Fanuc TP program (LS listing): DISTI_CADC_V7.LS

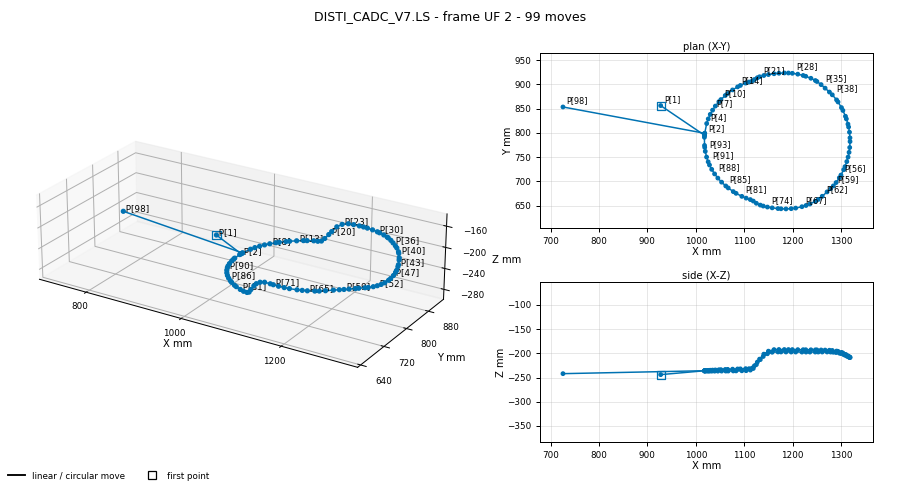
[picture p0: tool path of DISTI_CADC_V7.LS in frame UF 2, 99 of 99 moves have a stored position in this frame; points joined in program order, loops and branches not executed]
/PROG  DISTI_CADC_V7
/ATTR
OWNER		= MNEDITOR;
COMMENT		= "WeldPRO Auto-Gen";
PROG_SIZE	= 7109;
CREATE		= DATE 26-07-21  TIME 18:28:40;
MODIFIED	= DATE 26-07-21  TIME 18:47:32;
FILE_NAME	= DISTI_CA;
VERSION		= 0;
LINE_COUNT	= 113;
MEMORY_SIZE	= 7429;
PROTECT		= READ_WRITE;
TCD:  STACK_SIZE	= 0,
      TASK_PRIORITY	= 50,
      TIME_SLICE	= 0,
      BUSY_LAMP_OFF	= 0,
      ABORT_REQUEST	= 0,
      PAUSE_REQUEST	= 0;
DEFAULT_GROUP	= 1,*,*,*,*;
CONTROL_CODE	= 00000000 00000000;
/APPL
/MN
   1:  !WeldPRO Auto-Generated TPP ;
   2:  !Tor XL_176 _2, Feature1 ;
   3:   ;
   4:  UFRAME_NUM=2 ;
   5:  UTOOL_NUM=2 ;
   6:L P[1] 100mm/sec FINE    ;
   7:   ;
   8:  !Segment1 ;
   9:L P[2] 100mm/sec FINE    ;
  10:  CALL LASER_OFF    ;
  11:   ;
  12:L P[99] R[23:moving]mm/sec CNT100    ;
  13:   ;
  14:L P[3] R[23:moving]mm/sec CNT100    ;
  15:L P[4] R[23:moving]mm/sec CNT100    ;
  16:L P[5] R[23:moving]mm/sec CNT100    ;
  17:L P[6] R[23:moving]mm/sec CNT100    ;
  18:L P[7] R[23:moving]mm/sec CNT100    ;
  19:L P[8] R[23:moving]mm/sec CNT100    ;
  20:L P[9] R[23:moving]mm/sec CNT100    ;
  21:L P[10] R[23:moving]mm/sec CNT100    ;
  22:L P[11] R[23:moving]mm/sec CNT100    ;
  23:L P[12] R[23:moving]mm/sec CNT100    ;
  24:L P[13] R[23:moving]mm/sec CNT100    ;
  25:L P[14] R[23:moving]mm/sec CNT100    ;
  26:L P[15] R[23:moving]mm/sec CNT100    ;
  27:L P[16] R[23:moving]mm/sec CNT100    ;
  28:L P[17] R[23:moving]mm/sec CNT100    ;
  29:L P[18] R[23:moving]mm/sec CNT100    ;
  30:L P[19] R[23:moving]mm/sec CNT100    ;
  31:L P[20] R[23:moving]mm/sec CNT100    ;
  32:L P[21] R[23:moving]mm/sec CNT100    ;
  33:L P[22] R[23:moving]mm/sec CNT100    ;
  34:L P[23] R[23:moving]mm/sec CNT100    ;
  35:L P[24] R[23:moving]mm/sec CNT100    ;
  36:L P[25] R[23:moving]mm/sec CNT100    ;
  37:L P[26] R[23:moving]mm/sec CNT100    ;
  38:L P[27] R[23:moving]mm/sec CNT100    ;
  39:L P[28] R[23:moving]mm/sec CNT100    ;
  40:L P[29] R[23:moving]mm/sec CNT100    ;
  41:L P[30] R[23:moving]mm/sec CNT100    ;
  42:L P[31] R[23:moving]mm/sec CNT100    ;
  43:L P[32] R[23:moving]mm/sec CNT100    ;
  44:L P[33] R[23:moving]mm/sec CNT100    ;
  45:L P[34] R[23:moving]mm/sec CNT100    ;
  46:L P[35] R[23:moving]mm/sec CNT100    ;
  47:L P[36] R[23:moving]mm/sec CNT100    ;
  48:L P[37] R[23:moving]mm/sec CNT100    ;
  49:L P[38] R[23:moving]mm/sec CNT100    ;
  50:L P[39] R[23:moving]mm/sec CNT100    ;
  51:L P[40] R[23:moving]mm/sec CNT100    ;
  52:L P[41] R[23:moving]mm/sec CNT100    ;
  53:L P[42] R[23:moving]mm/sec CNT100    ;
  54:L P[43] R[23:moving]mm/sec CNT100    ;
  55:L P[44] R[23:moving]mm/sec CNT100    ;
  56:L P[45] R[23:moving]mm/sec CNT100    ;
  57:L P[46] R[23:moving]mm/sec CNT100    ;
  58:L P[47] R[23:moving]mm/sec CNT100    ;
  59:L P[48] R[23:moving]mm/sec CNT100    ;
  60:L P[49] R[23:moving]mm/sec CNT100    ;
  61:L P[50] R[23:moving]mm/sec CNT100    ;
  62:L P[51] R[23:moving]mm/sec CNT100    ;
  63:L P[52] R[23:moving]mm/sec CNT100    ;
  64:L P[53] R[23:moving]mm/sec CNT100    ;
  65:L P[54] R[23:moving]mm/sec CNT100    ;
  66:L P[55] R[23:moving]mm/sec CNT100    ;
  67:L P[56] R[23:moving]mm/sec CNT100    ;
  68:L P[57] R[23:moving]mm/sec CNT100    ;
  69:L P[58] R[23:moving]mm/sec CNT100    ;
  70:L P[59] R[23:moving]mm/sec CNT100    ;
  71:L P[60] R[23:moving]mm/sec CNT100    ;
  72:L P[61] R[23:moving]mm/sec CNT100    ;
  73:L P[62] R[23:moving]mm/sec CNT100    ;
  74:L P[63] R[23:moving]mm/sec CNT100    ;
  75:L P[64] R[23:moving]mm/sec CNT100    ;
  76:L P[65] R[23:moving]mm/sec CNT100    ;
  77:L P[66] R[23:moving]mm/sec CNT100    ;
  78:L P[67] R[23:moving]mm/sec CNT100    ;
  79:L P[68] R[23:moving]mm/sec CNT100    ;
  80:L P[69] R[23:moving]mm/sec CNT100    ;
  81:L P[70] R[23:moving]mm/sec CNT100    ;
  82:L P[71] R[23:moving]mm/sec CNT100    ;
  83:L P[72] R[23:moving]mm/sec CNT100    ;
  84:L P[73] R[23:moving]mm/sec CNT100    ;
  85:L P[74] R[23:moving]mm/sec CNT100    ;
  86:L P[75] R[23:moving]mm/sec CNT100    ;
  87:L P[76] R[23:moving]mm/sec CNT100    ;
  88:L P[77] R[23:moving]mm/sec CNT100    ;
  89:L P[78] R[23:moving]mm/sec CNT100    ;
  90:L P[79] R[23:moving]mm/sec CNT100    ;
  91:L P[80] R[23:moving]mm/sec CNT100    ;
  92:L P[81] R[23:moving]mm/sec CNT100    ;
  93:L P[82] R[23:moving]mm/sec CNT100    ;
  94:L P[83] R[23:moving]mm/sec CNT100    ;
  95:L P[84] R[23:moving]mm/sec CNT100    ;
  96:L P[85] R[23:moving]mm/sec CNT100    ;
  97:L P[86] R[23:moving]mm/sec CNT100    ;
  98:L P[87] R[23:moving]mm/sec CNT100    ;
  99:L P[88] R[23:moving]mm/sec CNT100    ;
 100:L P[89] R[23:moving]mm/sec CNT100    ;
 101:L P[90] R[23:moving]mm/sec CNT100    ;
 102:L P[91] R[23:moving]mm/sec CNT100    ;
 103:L P[92] R[23:moving]mm/sec CNT100    ;
 104:L P[93] R[23:moving]mm/sec CNT100    ;
 105:L P[94] R[23:moving]mm/sec CNT100    ;
 106:L P[95] R[23:moving]mm/sec CNT100    ;
 107:L P[96] R[23:moving]mm/sec CNT100    ;
 108:L P[97] R[23:moving]mm/sec FINE    ;
 109:  CALL LASER_OFF    ;
 110:   ;
 111:  !Feature Retreat ;
 112:L P[98] 100mm/sec FINE    ;
 113:  CALL ROTATE    ;
/POS
P[1]{
   GP1:
	UF : 2, UT : 2,		CONFIG : 'F D T, 0, 0, 0',
	X =   927.346  mm,	Y =   856.354  mm,	Z =  -244.034  mm,
	W =  -106.482 deg,	P =   -15.198 deg,	R =    86.345 deg
};
P[2]{
   GP1:
	UF : 2, UT : 2,		CONFIG : 'F D T, 0, 0, 0',
	X =  1017.889  mm,	Y =   795.080  mm,	Z =  -236.060  mm,
	W =  -106.491 deg,	P =   -15.193 deg,	R =    86.327 deg
};
P[3]{
   GP1:
	UF : 2, UT : 2,		CONFIG : 'F D T, 0, 0, 0',
	X =  1018.277  mm,	Y =   799.191  mm,	Z =  -235.971  mm,
	W =  -106.495 deg,	P =   -15.194 deg,	R =    86.332 deg
};
P[4]{
   GP1:
	UF : 2, UT : 2,		CONFIG : 'F D T, 0, 0, 0',
	X =  1022.296  mm,	Y =   819.337  mm,	Z =  -235.500  mm,
	W =  -106.425 deg,	P =   -15.445 deg,	R =    76.281 deg
};
P[5]{
   GP1:
	UF : 2, UT : 2,		CONFIG : 'F D T, 0, 0, 0',
	X =  1025.521  mm,	Y =   828.846  mm,	Z =  -235.241  mm,
	W =  -106.381 deg,	P =   -15.559 deg,	R =    71.464 deg
};
P[6]{
   GP1:
	UF : 2, UT : 2,		CONFIG : 'F D T, 0, 0, 0',
	X =  1029.666  mm,	Y =   838.199  mm,	Z =  -234.962  mm,
	W =  -106.310 deg,	P =   -15.698 deg,	R =    65.272 deg
};
P[7]{
   GP1:
	UF : 2, UT : 2,		CONFIG : 'F D T, 0, 0, 0',
	X =  1034.494  mm,	Y =   846.923  mm,	Z =  -234.669  mm,
	W =  -106.251 deg,	P =   -15.795 deg,	R =    60.811 deg
};
P[8]{
   GP1:
	UF : 2, UT : 2,		CONFIG : 'F D T, 0, 0, 0',
	X =  1040.175  mm,	Y =   855.353  mm,	Z =  -234.358  mm,
	W =  -106.174 deg,	P =   -15.897 deg,	R =    55.794 deg
};
P[9]{
   GP1:
	UF : 2, UT : 2,		CONFIG : 'F D T, 0, 0, 0',
	X =  1047.451  mm,	Y =   864.304  mm,	Z =  -233.991  mm,
	W =  -106.090 deg,	P =   -15.988 deg,	R =    50.970 deg
};
P[10]{
   GP1:
	UF : 2, UT : 2,		CONFIG : 'F D T, 0, 0, 0',
	X =  1051.689  mm,	Y =   868.820  mm,	Z =  -233.793  mm,
	W =  -106.027 deg,	P =   -16.056 deg,	R =    47.314 deg
};
P[11]{
   GP1:
	UF : 2, UT : 2,		CONFIG : 'F D T, 0, 0, 0',
	X =  1060.630  mm,	Y =   877.184  mm,	Z =  -233.387  mm,
	W =  -105.939 deg,	P =   -16.126 deg,	R =    42.935 deg
};
P[12]{
   GP1:
	UF : 2, UT : 2,		CONFIG : 'F D T, 0, 0, 0',
	X =  1065.640  mm,	Y =   881.308  mm,	Z =  -233.171  mm,
	W =  -105.872 deg,	P =   -16.175 deg,	R =    39.733 deg
};
P[13]{
   GP1:
	UF : 2, UT : 2,		CONFIG : 'F D T, 0, 0, 0',
	X =  1075.744  mm,	Y =   888.688  mm,	Z =  -232.750  mm,
	W =  -105.783 deg,	P =   -16.243 deg,	R =    35.484 deg
};
P[14]{
   GP1:
	UF : 2, UT : 2,		CONFIG : 'F D T, 0, 0, 0',
	X =  1086.136  mm,	Y =   894.999  mm,	Z =  -232.338  mm,
	W =  -105.683 deg,	P =   -16.290 deg,	R =    31.072 deg
};
P[15]{
   GP1:
	UF : 2, UT : 2,		CONFIG : 'F D T, 0, 0, 0',
	X =  1091.851  mm,	Y =   897.963  mm,	Z =  -232.125  mm,
	W =  -105.584 deg,	P =   -16.329 deg,	R =    26.914 deg
};
P[16]{
   GP1:
	UF : 2, UT : 2,		CONFIG : 'F D T, 0, 0, 0',
	X =  1102.710  mm,	Y =   902.806  mm,	Z =  -231.724  mm,
	W =  -105.545 deg,	P =   -16.341 deg,	R =    25.103 deg
};
P[17]{
   GP1:
	UF : 2, UT : 2,		CONFIG : 'F D T, 0, 0, 0',
	X =  1109.763  mm,	Y =   905.007  mm,	Z =  -231.762  mm,
	W =  -115.468 deg,	P =   -16.090 deg,	R =    30.046 deg
};
P[18]{
   GP1:
	UF : 2, UT : 2,		CONFIG : 'F D T, 0, 0, 0',
	X =  1116.013  mm,	Y =   906.877  mm,	Z =  -230.586  mm,
	W =  -126.721 deg,	P =   -15.366 deg,	R =    26.538 deg
};
P[19]{
   GP1:
	UF : 2, UT : 2,		CONFIG : 'F D T, 0, 0, 0',
	X =  1120.858  mm,	Y =   910.112  mm,	Z =  -225.766  mm,
	W =  -119.393 deg,	P =   -15.981 deg,	R =    16.221 deg
};
P[20]{
   GP1:
	UF : 2, UT : 2,		CONFIG : 'F D T, 0, 0, 0',
	X =  1126.832  mm,	Y =   913.808  mm,	Z =  -218.133  mm,
	W =  -115.329 deg,	P =   -16.208 deg,	R =    11.788 deg
};
P[21]{
   GP1:
	UF : 2, UT : 2,		CONFIG : 'F D T, 0, 0, 0',
	X =  1131.495  mm,	Y =   915.872  mm,	Z =  -212.049  mm,
	W =  -112.690 deg,	P =   -16.313 deg,	R =     9.687 deg
};
P[22]{
   GP1:
	UF : 2, UT : 2,		CONFIG : 'F D T, 0, 0, 0',
	X =  1140.206  mm,	Y =   918.445  mm,	Z =  -201.776  mm,
	W =  -110.089 deg,	P =   -16.384 deg,	R =     9.676 deg
};
P[23]{
   GP1:
	UF : 2, UT : 2,		CONFIG : 'F D T, 0, 0, 0',
	X =  1149.741  mm,	Y =   920.397  mm,	Z =  -195.589  mm,
	W =  -107.448 deg,	P =   -16.428 deg,	R =     8.430 deg
};
P[24]{
   GP1:
	UF : 2, UT : 2,		CONFIG : 'F D T, 0, 0, 0',
	X =  1161.315  mm,	Y =   922.076  mm,	Z =  -192.410  mm,
	W =  -105.451 deg,	P =   -16.442 deg,	R =     6.850 deg
};
P[25]{
   GP1:
	UF : 2, UT : 2,		CONFIG : 'F D T, 0, 0, 0',
	X =  1171.380  mm,	Y =   923.106  mm,	Z =  -192.191  mm,
	W =  -104.865 deg,	P =   -16.444 deg,	R =     5.674 deg
};
P[26]{
   GP1:
	UF : 2, UT : 2,		CONFIG : 'F D T, 0, 0, 0',
	X =  1182.566  mm,	Y =   923.704  mm,	Z =  -192.249  mm,
	W =  -104.885 deg,	P =   -16.444 deg,	R =     3.732 deg
};
P[27]{
   GP1:
	UF : 2, UT : 2,		CONFIG : 'F D T, 0, 0, 0',
	X =  1191.043  mm,	Y =   923.608  mm,	Z =  -192.305  mm,
	W =  -104.928 deg,	P =   -16.440 deg,	R =     -.482 deg
};
P[28]{
   GP1:
	UF : 2, UT : 2,		CONFIG : 'F D T, 0, 0, 0',
	X =  1199.100  mm,	Y =   922.988  mm,	Z =  -192.368  mm,
	W =  -104.977 deg,	P =   -16.425 deg,	R =    -5.295 deg
};
P[29]{
   GP1:
	UF : 2, UT : 2,		CONFIG : 'F D T, 0, 0, 0',
	X =  1210.327  mm,	Y =   921.245  mm,	Z =  -192.471  mm,
	W =  -105.026 deg,	P =   -16.401 deg,	R =   -10.039 deg
};
P[30]{
   GP1:
	UF : 2, UT : 2,		CONFIG : 'F D T, 0, 0, 0',
	X =  1221.437  mm,	Y =   918.518  mm,	Z =  -192.590  mm,
	W =  -105.069 deg,	P =   -16.371 deg,	R =   -14.284 deg
};
P[31]{
   GP1:
	UF : 2, UT : 2,		CONFIG : 'F D T, 0, 0, 0',
	X =  1226.752  mm,	Y =   916.839  mm,	Z =  -192.653  mm,
	W =  -105.112 deg,	P =   -16.334 deg,	R =   -18.515 deg
};
P[32]{
   GP1:
	UF : 2, UT : 2,		CONFIG : 'F D T, 0, 0, 0',
	X =  1237.398  mm,	Y =   912.751  mm,	Z =  -192.794  mm,
	W =  -105.156 deg,	P =   -16.287 deg,	R =   -22.931 deg
};
P[33]{
   GP1:
	UF : 2, UT : 2,		CONFIG : 'F D T, 0, 0, 0',
	X =  1246.694  mm,	Y =   908.067  mm,	Z =  -192.936  mm,
	W =  -105.219 deg,	P =   -16.204 deg,	R =   -29.417 deg
};
P[34]{
   GP1:
	UF : 2, UT : 2,		CONFIG : 'F D T, 0, 0, 0',
	X =  1249.746  mm,	Y =   906.136  mm,	Z =  -192.994  mm,
	W =  -105.326 deg,	P =   -16.106 deg,	R =   -35.234 deg
};
P[35]{
   GP1:
	UF : 2, UT : 2,		CONFIG : 'F D T, 0, 0, 0',
	X =  1258.465  mm,	Y =   899.675  mm,	Z =  -193.157  mm,
	W =  -105.307 deg,	P =   -16.055 deg,	R =   -38.974 deg
};
P[36]{
   GP1:
	UF : 2, UT : 2,		CONFIG : 'F D T, 0, 0, 0',
	X =  1266.694  mm,	Y =   892.374  mm,	Z =  -193.348  mm,
	W =  -105.304 deg,	P =   -16.061 deg,	R =   -38.624 deg
};
P[37]{
   GP1:
	UF : 2, UT : 2,		CONFIG : 'F D T, 0, 0, 0',
	X =  1275.636  mm,	Y =   884.289  mm,	Z =  -193.707  mm,
	W =  -105.460 deg,	P =   -15.949 deg,	R =   -44.737 deg
};
P[38]{
   GP1:
	UF : 2, UT : 2,		CONFIG : 'F D T, 0, 0, 0',
	X =  1281.534  mm,	Y =   878.597  mm,	Z =  -194.154  mm,
	W =  -105.652 deg,	P =   -15.892 deg,	R =   -47.603 deg
};
P[39]{
   GP1:
	UF : 2, UT : 2,		CONFIG : 'F D T, 0, 0, 0',
	X =  1290.405  mm,	Y =   868.154  mm,	Z =  -195.366  mm,
	W =  -106.194 deg,	P =   -15.794 deg,	R =   -52.149 deg
};
P[40]{
   GP1:
	UF : 2, UT : 2,		CONFIG : 'F D T, 0, 0, 0',
	X =  1293.358  mm,	Y =   863.881  mm,	Z =  -196.009  mm,
	W =  -106.906 deg,	P =   -15.690 deg,	R =   -56.548 deg
};
P[41]{
   GP1:
	UF : 2, UT : 2,		CONFIG : 'F D T, 0, 0, 0',
	X =  1300.478  mm,	Y =   852.200  mm,	Z =  -198.134  mm,
	W =  -107.559 deg,	P =   -15.603 deg,	R =   -60.015 deg
};
P[42]{
   GP1:
	UF : 2, UT : 2,		CONFIG : 'F D T, 0, 0, 0',
	X =  1303.428  mm,	Y =   846.403  mm,	Z =  -199.394  mm,
	W =  -108.250 deg,	P =   -15.507 deg,	R =   -63.574 deg
};
P[43]{
   GP1:
	UF : 2, UT : 2,		CONFIG : 'F D T, 0, 0, 0',
	X =  1308.723  mm,	Y =   834.279  mm,	Z =  -202.322  mm,
	W =  -109.123 deg,	P =   -15.380 deg,	R =   -68.091 deg
};
P[44]{
   GP1:
	UF : 2, UT : 2,		CONFIG : 'F D T, 0, 0, 0',
	X =  1310.604  mm,	Y =   828.898  mm,	Z =  -203.468  mm,
	W =  -109.894 deg,	P =   -15.253 deg,	R =   -72.476 deg
};
P[45]{
   GP1:
	UF : 2, UT : 2,		CONFIG : 'F D T, 0, 0, 0',
	X =  1313.867  mm,	Y =   818.113  mm,	Z =  -205.461  mm,
	W =  -110.258 deg,	P =   -15.184 deg,	R =   -74.873 deg
};
P[46]{
   GP1:
	UF : 2, UT : 2,		CONFIG : 'F D T, 0, 0, 0',
	X =  1315.235  mm,	Y =   812.168  mm,	Z =  -206.340  mm,
	W =  -110.625 deg,	P =   -15.098 deg,	R =   -77.924 deg
};
P[47]{
   GP1:
	UF : 2, UT : 2,		CONFIG : 'F D T, 0, 0, 0',
	X =  1317.027  mm,	Y =   801.431  mm,	Z =  -207.574  mm,
	W =  -111.046 deg,	P =   -14.958 deg,	R =   -82.908 deg
};
P[48]{
   GP1:
	UF : 2, UT : 2,		CONFIG : 'F D T, 0, 0, 0',
	X =  1318.033  mm,	Y =   789.801  mm,	Z =  -208.385  mm,
	W =  -111.160 deg,	P =   -14.266 deg,	R =   -88.178 deg
};
P[49]{
   GP1:
	UF : 2, UT : 2,		CONFIG : 'F D T, 0, 0, 0',
	X =  1318.168  mm,	Y =   782.182  mm,	Z =  -208.610  mm,
	W =  -111.104 deg,	P =   -14.627 deg,	R =   -91.603 deg
};
P[50]{
   GP1:
	UF : 2, UT : 2,		CONFIG : 'F D T, 0, 0, 0',
	X =  1317.501  mm,	Y =   769.857  mm,	Z =  -208.488  mm,
	W =  -110.785 deg,	P =   -15.101 deg,	R =   -96.403 deg
};
P[51]{
   GP1:
	UF : 2, UT : 2,		CONFIG : 'F D T, 0, 0, 0',
	X =  1316.168  mm,	Y =   759.918  mm,	Z =  -207.950  mm,
	W =  -110.276 deg,	P =   -14.535 deg,	R =  -100.836 deg
};
P[52]{
   GP1:
	UF : 2, UT : 2,		CONFIG : 'F D T, 0, 0, 0',
	X =  1314.124  mm,	Y =   750.096  mm,	Z =  -207.025  mm,
	W =  -109.635 deg,	P =   -14.447 deg,	R =  -105.265 deg
};
P[53]{
   GP1:
	UF : 2, UT : 2,		CONFIG : 'F D T, 0, 0, 0',
	X =  1311.503  mm,	Y =   740.771  mm,	Z =  -205.798  mm,
	W =  -109.103 deg,	P =   -14.384 deg,	R =  -108.504 deg
};
P[54]{
   GP1:
	UF : 2, UT : 2,		CONFIG : 'F D T, 0, 0, 0',
	X =  1307.757  mm,	Y =   730.358  mm,	Z =  -204.011  mm,
	W =  -108.392 deg,	P =   -14.307 deg,	R =  -112.625 deg
};
P[55]{
   GP1:
	UF : 2, UT : 2,		CONFIG : 'F D T, 0, 0, 0',
	X =  1305.065  mm,	Y =   724.102  mm,	Z =  -202.728  mm,
	W =  -107.773 deg,	P =   -14.241 deg,	R =  -116.139 deg
};
P[56]{
   GP1:
	UF : 2, UT : 2,		CONFIG : 'F D T, 0, 0, 0',
	X =  1299.418  mm,	Y =   712.954  mm,	Z =  -200.557  mm,
	W =  -106.932 deg,	P =   -14.149 deg,	R =  -121.162 deg
};
P[57]{
   GP1:
	UF : 2, UT : 2,		CONFIG : 'F D T, 0, 0, 0',
	X =  1296.056  mm,	Y =   707.282  mm,	Z =  -199.652  mm,
	W =  -106.269 deg,	P =   -14.066 deg,	R =  -125.698 deg
};
P[58]{
   GP1:
	UF : 2, UT : 2,		CONFIG : 'F D T, 0, 0, 0',
	X =  1289.374  mm,	Y =   697.456  mm,	Z =  -198.422  mm,
	W =  -105.781 deg,	P =   -13.988 deg,	R =  -130.143 deg
};
P[59]{
   GP1:
	UF : 2, UT : 2,		CONFIG : 'F D T, 0, 0, 0',
	X =  1283.723  mm,	Y =   690.590  mm,	Z =  -197.821  mm,
	W =  -105.502 deg,	P =   -13.914 deg,	R =  -134.519 deg
};
P[60]{
   GP1:
	UF : 2, UT : 2,		CONFIG : 'F D T, 0, 0, 0',
	X =  1278.164  mm,	Y =   684.885  mm,	Z =  -197.494  mm,
	W =  -105.438 deg,	P =   -13.851 deg,	R =  -138.498 deg
};
P[61]{
   GP1:
	UF : 2, UT : 2,		CONFIG : 'F D T, 0, 0, 0',
	X =  1270.775  mm,	Y =   678.212  mm,	Z =  -197.291  mm,
	W =  -105.428 deg,	P =   -13.829 deg,	R =  -139.977 deg
};
P[62]{
   GP1:
	UF : 2, UT : 2,		CONFIG : 'F D T, 0, 0, 0',
	X =  1260.749  mm,	Y =   669.204  mm,	Z =  -197.348  mm,
	W =  -105.443 deg,	P =   -13.863 deg,	R =  -137.727 deg
};
P[63]{
   GP1:
	UF : 2, UT : 2,		CONFIG : 'F D T, 0, 0, 0',
	X =  1252.575  mm,	Y =   662.699  mm,	Z =  -197.405  mm,
	W =  -105.373 deg,	P =   -13.729 deg,	R =  -147.436 deg
};
P[64]{
   GP1:
	UF : 2, UT : 2,		CONFIG : 'F D T, 0, 0, 0',
	X =  1246.362  mm,	Y =   658.782  mm,	Z =  -197.421  mm,
	W =  -105.298 deg,	P =   -13.637 deg,	R =  -156.529 deg
};
P[65]{
   GP1:
	UF : 2, UT : 2,		CONFIG : 'F D T, 0, 0, 0',
	X =  1235.369  mm,	Y =   653.232  mm,	Z =  -197.454  mm,
	W =  -105.278 deg,	P =   -13.619 deg,	R =  -158.873 deg
};
P[66]{
   GP1:
	UF : 2, UT : 2,		CONFIG : 'F D T, 0, 0, 0',
	X =  1227.306  mm,	Y =   650.188  mm,	Z =  -197.457  mm,
	W =  -105.242 deg,	P =   -13.593 deg,	R =  -162.872 deg
};
P[67]{
   GP1:
	UF : 2, UT : 2,		CONFIG : 'F D T, 0, 0, 0',
	X =  1218.912  mm,	Y =   647.653  mm,	Z =  -197.449  mm,
	W =  -105.204 deg,	P =   -13.573 deg,	R =  -166.917 deg
};
P[68]{
   GP1:
	UF : 2, UT : 2,		CONFIG : 'F D T, 0, 0, 0',
	X =  1205.982  mm,	Y =   644.800  mm,	Z =  -197.421  mm,
	W =  -105.160 deg,	P =   -13.560 deg,	R =  -171.451 deg
};
P[69]{
   GP1:
	UF : 2, UT : 2,		CONFIG : 'F D T, 0, 0, 0',
	X =  1196.678  mm,	Y =   643.604  mm,	Z =  -197.386  mm,
	W =  -105.114 deg,	P =   -13.556 deg,	R =  -176.195 deg
};
P[70]{
   GP1:
	UF : 2, UT : 2,		CONFIG : 'F D T, 0, 0, 0',
	X =  1185.921  mm,	Y =   643.103  mm,	Z =  -197.326  mm,
	W =  -105.069 deg,	P =   -13.561 deg,	R =   179.311 deg
};
P[71]{
   GP1:
	UF : 2, UT : 2,		CONFIG : 'F D T, 0, 0, 0',
	X =  1175.641  mm,	Y =   643.412  mm,	Z =  -197.255  mm,
	W =  -105.038 deg,	P =   -13.569 deg,	R =   176.231 deg
};
P[72]{
   GP1:
	UF : 2, UT : 2,		CONFIG : 'F D T, 0, 0, 0',
	X =  1169.439  mm,	Y =   643.884  mm,	Z =  -197.231  mm,
	W =  -105.170 deg,	P =   -13.572 deg,	R =   175.317 deg
};
P[73]{
   GP1:
	UF : 2, UT : 2,		CONFIG : 'F D T, 0, 0, 0',
	X =  1157.478  mm,	Y =   645.299  mm,	Z =  -197.840  mm,
	W =  -106.961 deg,	P =   -13.569 deg,	R =   174.549 deg
};
P[74]{
   GP1:
	UF : 2, UT : 2,		CONFIG : 'F D T, 0, 0, 0',
	X =  1147.662  mm,	Y =   646.981  mm,	Z =  -200.943  mm,
	W =  -109.346 deg,	P =   -13.539 deg,	R =   174.478 deg
};
P[75]{
   GP1:
	UF : 2, UT : 2,		CONFIG : 'F D T, 0, 0, 0',
	X =  1139.035  mm,	Y =   649.035  mm,	Z =  -206.577  mm,
	W =  -112.145 deg,	P =   -13.468 deg,	R =   175.272 deg
};
P[76]{
   GP1:
	UF : 2, UT : 2,		CONFIG : 'F D T, 0, 0, 0',
	X =  1132.964  mm,	Y =   651.006  mm,	Z =  -213.027  mm,
	W =  -114.824 deg,	P =   -13.371 deg,	R =   175.449 deg
};
P[77]{
   GP1:
	UF : 2, UT : 2,		CONFIG : 'F D T, 0, 0, 0',
	X =  1124.814  mm,	Y =   654.759  mm,	Z =  -223.318  mm,
	W =  -120.114 deg,	P =   -13.109 deg,	R =   172.293 deg
};
P[78]{
   GP1:
	UF : 2, UT : 2,		CONFIG : 'F D T, 0, 0, 0',
	X =  1118.504  mm,	Y =   659.310  mm,	Z =  -231.322  mm,
	W =  -126.491 deg,	P =   -12.649 deg,	R =   168.032 deg
};
P[79]{
   GP1:
	UF : 2, UT : 2,		CONFIG : 'F D T, 0, 0, 0',
	X =  1112.437  mm,	Y =   662.363  mm,	Z =  -234.682  mm,
	W =  -119.899 deg,	P =   -13.263 deg,	R =   157.916 deg
};
P[80]{
   GP1:
	UF : 2, UT : 2,		CONFIG : 'F D T, 0, 0, 0',
	X =  1103.727  mm,	Y =   665.395  mm,	Z =  -235.889  mm,
	W =  -106.920 deg,	P =   -13.744 deg,	R =   154.284 deg
};
P[81]{
   GP1:
	UF : 2, UT : 2,		CONFIG : 'F D T, 0, 0, 0',
	X =  1094.873  mm,	Y =   669.053  mm,	Z =  -236.088  mm,
	W =  -105.725 deg,	P =   -13.738 deg,	R =   155.031 deg
};
P[82]{
   GP1:
	UF : 2, UT : 2,		CONFIG : 'F D T, 0, 0, 0',
	X =  1082.969  mm,	Y =   675.268  mm,	Z =  -236.338  mm,
	W =  -105.804 deg,	P =   -13.784 deg,	R =   151.515 deg
};
P[83]{
   GP1:
	UF : 2, UT : 2,		CONFIG : 'F D T, 0, 0, 0',
	X =  1077.181  mm,	Y =   678.862  mm,	Z =  -236.443  mm,
	W =  -105.884 deg,	P =   -13.836 deg,	R =   147.827 deg
};
P[84]{
   GP1:
	UF : 2, UT : 2,		CONFIG : 'F D T, 0, 0, 0',
	X =  1066.729  mm,	Y =   686.379  mm,	Z =  -236.616  mm,
	W =  -105.989 deg,	P =   -13.919 deg,	R =   142.627 deg
};
P[85]{
   GP1:
	UF : 2, UT : 2,		CONFIG : 'F D T, 0, 0, 0',
	X =  1061.717  mm,	Y =   690.490  mm,	Z =  -236.674  mm,
	W =  -106.066 deg,	P =   -13.990 deg,	R =   138.574 deg
};
P[86]{
   GP1:
	UF : 2, UT : 2,		CONFIG : 'F D T, 0, 0, 0',
	X =  1053.084  mm,	Y =   698.346  mm,	Z =  -236.726  mm,
	W =  -106.118 deg,	P =   -14.044 deg,	R =   135.639 deg
};
P[87]{
   GP1:
	UF : 2, UT : 2,		CONFIG : 'F D T, 0, 0, 0',
	X =  1045.340  mm,	Y =   706.715  mm,	Z =  -236.809  mm,
	W =  -106.192 deg,	P =   -14.130 deg,	R =   131.212 deg
};
P[88]{
   GP1:
	UF : 2, UT : 2,		CONFIG : 'F D T, 0, 0, 0',
	X =  1038.635  mm,	Y =   715.377  mm,	Z =  -236.868  mm,
	W =  -106.261 deg,	P =   -14.227 deg,	R =   126.545 deg
};
P[89]{
   GP1:
	UF : 2, UT : 2,		CONFIG : 'F D T, 0, 0, 0',
	X =  1032.687  mm,	Y =   724.747  mm,	Z =  -236.859  mm,
	W =  -106.325 deg,	P =   -14.335 deg,	R =   121.649 deg
};
P[90]{
   GP1:
	UF : 2, UT : 2,		CONFIG : 'F D T, 0, 0, 0',
	X =  1028.093  mm,	Y =   733.775  mm,	Z =  -236.812  mm,
	W =  -106.396 deg,	P =   -14.486 deg,	R =   115.073 deg
};
P[91]{
   GP1:
	UF : 2, UT : 2,		CONFIG : 'F D T, 0, 0, 0',
	X =  1025.370  mm,	Y =   740.318  mm,	Z =  -236.773  mm,
	W =  -106.437 deg,	P =   -14.604 deg,	R =   110.157 deg
};
P[92]{
   GP1:
	UF : 2, UT : 2,		CONFIG : 'F D T, 0, 0, 0',
	X =  1022.103  mm,	Y =   750.152  mm,	Z =  -236.722  mm,
	W =  -106.467 deg,	P =   -14.723 deg,	R =   105.309 deg
};
P[93]{
   GP1:
	UF : 2, UT : 2,		CONFIG : 'F D T, 0, 1, 0',
	X =  1019.394  mm,	Y =   761.936  mm,	Z =  -236.624  mm,
	W =  -106.486 deg,	P =   -14.842 deg,	R =   100.517 deg
};
P[94]{
   GP1:
	UF : 2, UT : 2,		CONFIG : 'F D T, 0, 1, 0',
	X =  1018.238  mm,	Y =   770.114  mm,	Z =  -236.509  mm,
	W =  -106.495 deg,	P =   -14.962 deg,	R =    95.763 deg
};
P[95]{
   GP1:
	UF : 2, UT : 2,		CONFIG : 'F D T, 0, 1, 0',
	X =  1017.859  mm,	Y =   774.098  mm,	Z =  -236.443  mm,
	W =  -106.506 deg,	P =   -15.000 deg,	R =    94.230 deg
};
P[96]{
   GP1:
	UF : 2, UT : 2,		CONFIG : 'F D T, 0, 1, 0',
	X =  1017.634  mm,	Y =   790.896  mm,	Z =  -236.145  mm,
	W =  -106.482 deg,	P =   -15.197 deg,	R =    86.402 deg
};
P[97]{
   GP1:
	UF : 2, UT : 2,		CONFIG : 'F D T, 0, 1, 0',
	X =  1018.276  mm,	Y =   799.188  mm,	Z =  -235.969  mm,
	W =  -106.482 deg,	P =   -15.198 deg,	R =    86.345 deg
};
P[98]{
   GP1:
	UF : 2, UT : 2,		CONFIG : 'F D T, 0, 1, 0',
	X =   725.689  mm,	Y =   853.506  mm,	Z =  -242.034  mm,
	W =  -106.487 deg,	P =   -15.200 deg,	R =    86.348 deg
};
P[99]{
   GP1:
	UF : 2, UT : 2,		CONFIG : 'F D T, 0, 0, 0',
	X =  1017.889  mm,	Y =   795.080  mm,	Z =  -236.060  mm,
	W =  -106.495 deg,	P =   -15.194 deg,	R =    86.332 deg
};
/END
